PROGRAM ReplaceAll
// Replaces all the instances of the input string with another string
// If In_StringToSearch := 'aaaaa123aaaaa123aaaaaaa123aaaaa123'
// In_StringToFind := '123'
// In_StringToReplace : = 'ABC'
// Then : OUT_StringToSearch := 'aaaaaABCaaaaaABCaaaaaaaABCaaaaaABC'
// Equivalent to CTRL + H
VAR_INPUT
	IN_StringToSearch	: T_MaxString;		// String to search : main string with instances we wish to replace
	IN_StringToFind		: STRING;			// String we are looking to find in the String_To_Seach
	IN_StringToReplace 	: STRING;			// String with which we want to replace the String To Find in String To Search
END_VAR

VAR_OUTPUT
	OUT_StringToSearch : T_MaxString;		// Output String
END_VAR

VAR
	KK: INT;
	Test_INT : INT;
END_VAR

OUT_StringToSearch := IN_StringToSearch;
FOR KK := 1 TO LEN(STR := OUT_StringToSearch) DO
	Test_INT := FIND(STR1 := OUT_StringToSearch, STR2 := IN_StringToFind);
	IF Test_INT > 0 THEN
		OUT_StringToSearch := REPLACE(STR1 := OUT_StringToSearch, STR2 := IN_StringToReplace, P := Test_INT, L := len(IN_StringToFind));
		KK := Test_Int;
	END_IF
END_FOR

END_PROGRAM

(* stored: Version 1.1.0.1, ProductVersion 3.1.4024.6
   POU ReplaceAll: Id {10a0049b-258e-4aee-bc6f-d4dcdb439021}, SpecialFunc None *)
